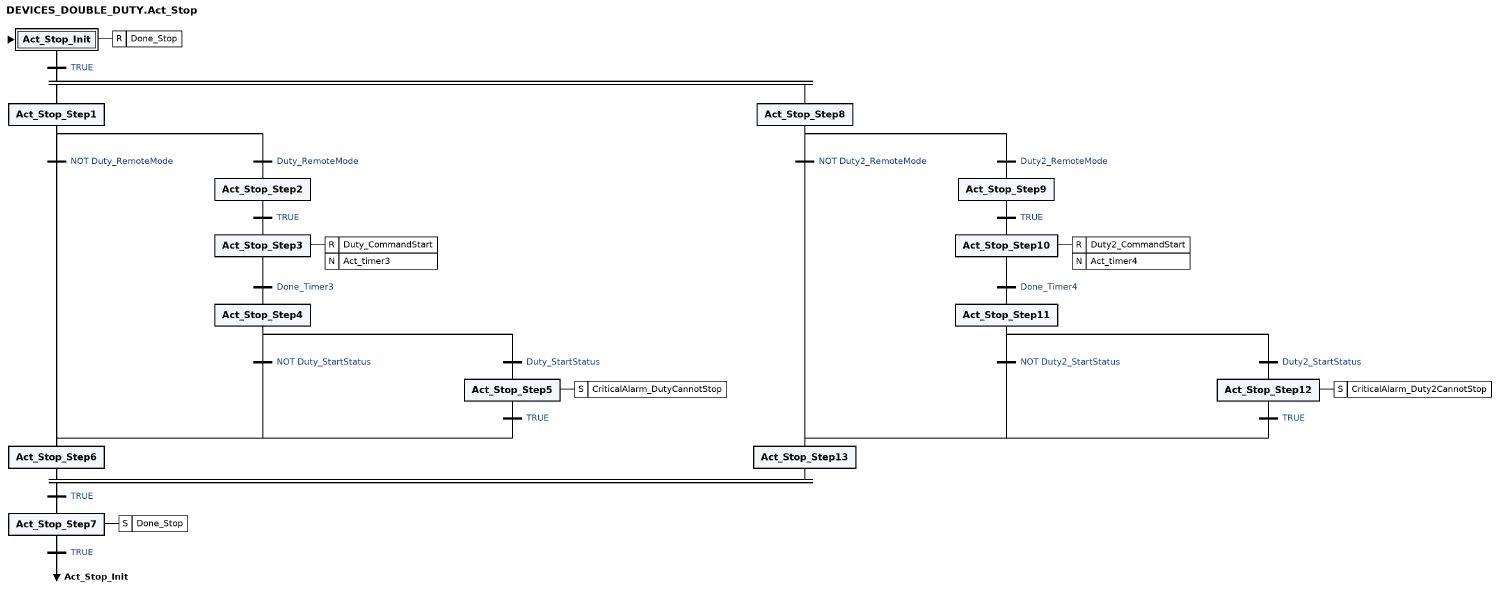
INITIAL_STEP Act_Stop_Init:
	Done_Stop(R);
END_STEP
TRANSITION FROM Act_Stop_Init TO (Act_Stop_Step1, Act_Stop_Step8) := TRUE;
END_TRANSITION
STEP Act_Stop_Step1:
END_STEP
TRANSITION FROM Act_Stop_Step1 TO Act_Stop_Step6 := NOT Duty_RemoteMode;
END_TRANSITION
TRANSITION FROM Act_Stop_Step1 TO Act_Stop_Step2 := Duty_RemoteMode;
END_TRANSITION
STEP Act_Stop_Step2:
END_STEP
TRANSITION FROM Act_Stop_Step2 TO Act_Stop_Step3 := TRUE;
END_TRANSITION
STEP Act_Stop_Step3:
	Duty_CommandStart(R);
	Act_timer3(N);
END_STEP
TRANSITION FROM Act_Stop_Step3 TO Act_Stop_Step4 := Done_Timer3;
END_TRANSITION
STEP Act_Stop_Step4:
END_STEP
TRANSITION FROM Act_Stop_Step4 TO Act_Stop_Step6 := NOT Duty_StartStatus;
END_TRANSITION
TRANSITION FROM Act_Stop_Step4 TO Act_Stop_Step5 := Duty_StartStatus;
END_TRANSITION
STEP Act_Stop_Step5:
	CriticalAlarm_DutyCannotStop(S);
END_STEP
TRANSITION FROM Act_Stop_Step5 TO Act_Stop_Step6 := TRUE;
END_TRANSITION
STEP Act_Stop_Step6:
END_STEP
STEP Act_Stop_Step8:
END_STEP
TRANSITION FROM Act_Stop_Step8 TO Act_Stop_Step13 := NOT Duty2_RemoteMode;
END_TRANSITION
TRANSITION FROM Act_Stop_Step8 TO Act_Stop_Step9 := Duty2_RemoteMode;
END_TRANSITION
STEP Act_Stop_Step9:
END_STEP
TRANSITION FROM Act_Stop_Step9 TO Act_Stop_Step10 := TRUE;
END_TRANSITION
STEP Act_Stop_Step10:
	Duty2_CommandStart(R);
	Act_timer4(N);
END_STEP
TRANSITION FROM Act_Stop_Step10 TO Act_Stop_Step11 := Done_Timer4;
END_TRANSITION
STEP Act_Stop_Step11:
END_STEP
TRANSITION FROM Act_Stop_Step11 TO Act_Stop_Step13 := NOT Duty2_StartStatus;
END_TRANSITION
TRANSITION FROM Act_Stop_Step11 TO Act_Stop_Step12 := Duty2_StartStatus;
END_TRANSITION
STEP Act_Stop_Step12:
	CriticalAlarm_Duty2CannotStop(S);
END_STEP
TRANSITION FROM Act_Stop_Step12 TO Act_Stop_Step13 := TRUE;
END_TRANSITION
STEP Act_Stop_Step13:
END_STEP
TRANSITION FROM (Act_Stop_Step6, Act_Stop_Step13) TO Act_Stop_Step7 := TRUE;
END_TRANSITION
STEP Act_Stop_Step7:
	Done_Stop(S);
END_STEP
TRANSITION FROM Act_Stop_Step7 TO Act_Stop_Init := TRUE;
END_TRANSITION
END_ACTION
ACTION Act_Timer:
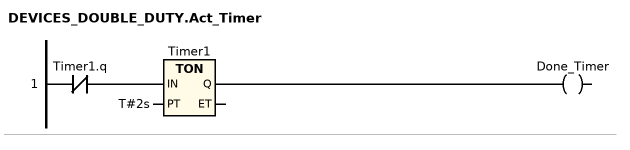
_LD_ (* Ladder Diagram *)
NETWORK 1
	[/Timer1.q] - Timer1:TON(IN: *, PT: T#2s) --- (Done_Timer)
_END_LD_
(* the same logic as Structured Text *)
(* Network 1 *)
Timer1(IN := NOT Timer1.q, PT := T#2s);
Done_Timer := Timer1.Q;
END_ACTION
ACTION Act_Timer2:
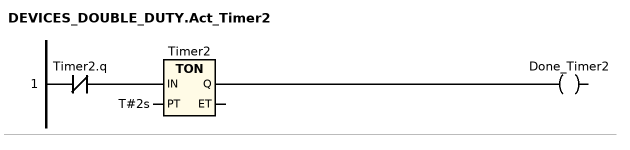
_LD_ (* Ladder Diagram *)
NETWORK 1
	[/Timer2.q] - Timer2:TON(IN: *, PT: T#2s) --- (Done_Timer2)
_END_LD_
(* the same logic as Structured Text *)
(* Network 1 *)
Timer2(IN := NOT Timer2.q, PT := T#2s);
Done_Timer2 := Timer2.Q;
END_ACTION
ACTION Act_Timer3:
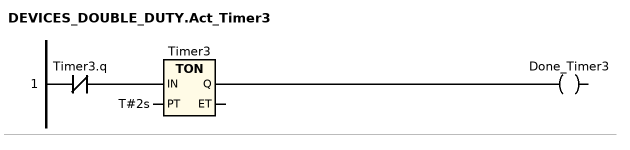
_LD_ (* Ladder Diagram *)
NETWORK 1
	[/Timer3.q] - Timer3:TON(IN: *, PT: T#2s) --- (Done_Timer3)
_END_LD_
(* the same logic as Structured Text *)
(* Network 1 *)
Timer3(IN := NOT Timer3.q, PT := T#2s);
Done_Timer3 := Timer3.Q;
END_ACTION
ACTION Act_Timer4:
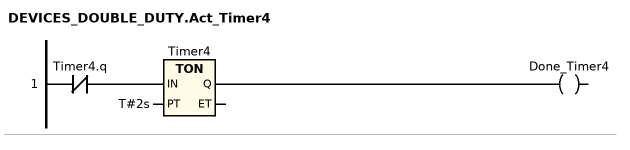
_LD_ (* Ladder Diagram *)
NETWORK 1
	[/Timer4.q] - Timer4:TON(IN: *, PT: T#2s) --- (Done_Timer4)
_END_LD_
(* the same logic as Structured Text *)
(* Network 1 *)
Timer4(IN := NOT Timer4.q, PT := T#2s);
Done_Timer4 := Timer4.Q;
END_ACTION

(* POU test, ST *)
FUNCTION_BLOCK test
VAR_INPUT
END_VAR
VAR_OUTPUT
END_VAR
VAR
	test : ARRAY [0..99] OF INT;
	x: INT;
END_VAR
(*
FOR x:= 0 TO 99 DO
test[x] := 99;
END_FOR
*);
END_FUNCTION_BLOCK

(* POU REUSE_WATER_SYS, SFC *)
FUNCTION_BLOCK REUSE_WATER_SYS
VAR_INPUT
END_VAR
VAR_OUTPUT
END_VAR
VAR
	VacumPump_AB : DEVICES_DUTY_STANDBY;
	LeadPump_AB : DEVICES_DOUBLE_DUTY;
	LeadPump_CD: DEVICES_DOUBLE_DUTY;
	JockeyPump_AB : DEVICES_DUTY_STANDBY;
	LSL308A AT%I*: BOOL;
	LSH308B AT%I*: BOOL;
	LSL308B AT%I*: BOOL;
	LSH308A AT%I*: BOOL;
	Done_Active: BOOL;
	XV101 AT%Q* : BOOL;
	XV102 AT%Q*: BOOL;
	Done_Vacum_Priming: BOOL;
	Done_On_Pump_Seq: BOOL;
	LSH406 AT%I*: BOOL;
	FSL101 AT%I*: BOOL;
	LSH405 AT%I*: BOOL;
	WaterPressureSensor: LREAL;
	Timer1: TON;
	done_TimerWaterPressure: BOOL;
	Reset_TimerWaterPressure: BOOL;
	WarningAlarm_HighPressure : BOOL;
	Done_stop: BOOL;
	RESET: BOOL;
END_VAR
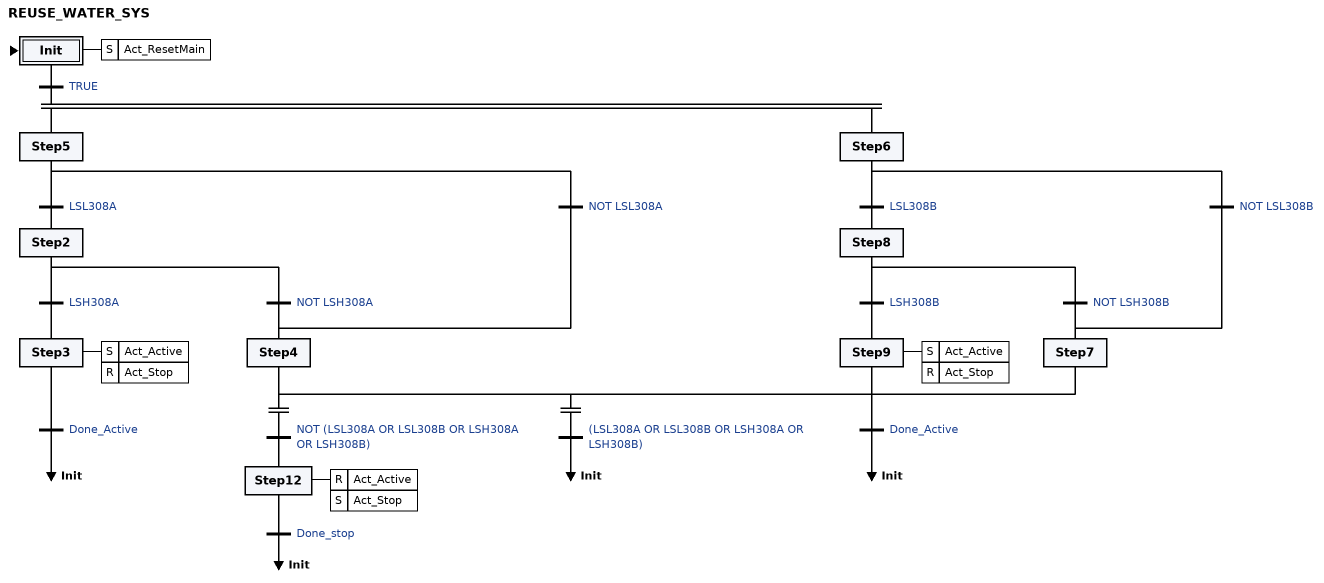
INITIAL_STEP Init:
	Act_ResetMain(S);
END_STEP
TRANSITION FROM Init TO (Step5, Step6) := TRUE;
END_TRANSITION
STEP Step5:
END_STEP
TRANSITION FROM Step5 TO Step2 := LSL308A;
END_TRANSITION
TRANSITION FROM Step5 TO Step4 := NOT LSL308A;
END_TRANSITION
STEP Step2:
END_STEP
TRANSITION FROM Step2 TO Step3 := LSH308A;
END_TRANSITION
TRANSITION FROM Step2 TO Step4 := NOT LSH308A;
END_TRANSITION
STEP Step3:
	Act_Active(S);
	Act_Stop(R);
END_STEP
TRANSITION FROM Step3 TO Init := Done_Active;
END_TRANSITION
STEP Step4:
END_STEP
STEP Step6:
END_STEP
TRANSITION FROM Step6 TO Step8 := LSL308B;
END_TRANSITION
TRANSITION FROM Step6 TO Step7 := NOT LSL308B;
END_TRANSITION
STEP Step8:
END_STEP
TRANSITION FROM Step8 TO Step9 := LSH308B;
END_TRANSITION
TRANSITION FROM Step8 TO Step7 := NOT LSH308B;
END_TRANSITION
STEP Step9:
	Act_Active(S);
	Act_Stop(R);
END_STEP
TRANSITION FROM Step9 TO Init := Done_Active;
END_TRANSITION
STEP Step7:
END_STEP
TRANSITION FROM (Step4, Step7) TO Step12 := NOT (LSL308A OR LSL308B OR LSH308A OR LSH308B);
END_TRANSITION
TRANSITION FROM (Step4, Step7) TO Init := (LSL308A OR LSL308B OR LSH308A OR LSH308B);
END_TRANSITION
STEP Step12:
	Act_Active(R);
	Act_Stop(S);
END_STEP
TRANSITION FROM Step12 TO Init := Done_stop;
END_TRANSITION
END_FUNCTION_BLOCK
ACTION Act_Active:
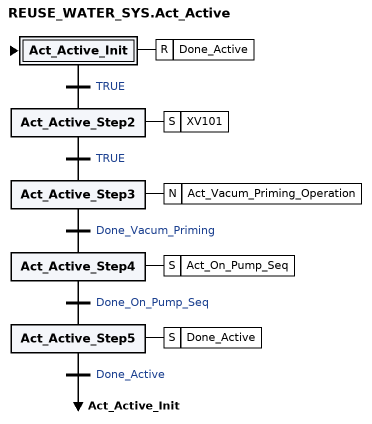
INITIAL_STEP Act_Active_Init:
	Done_Active(R);
END_STEP
TRANSITION FROM Act_Active_Init TO Act_Active_Step2 := TRUE;
END_TRANSITION
STEP Act_Active_Step2:
	XV101(S);
END_STEP
TRANSITION FROM Act_Active_Step2 TO Act_Active_Step3 := TRUE;
END_TRANSITION
STEP Act_Active_Step3:
	Act_Vacum_Priming_Operation(N);
END_STEP
TRANSITION FROM Act_Active_Step3 TO Act_Active_Step4 := Done_Vacum_Priming;
END_TRANSITION
STEP Act_Active_Step4:
	Act_On_Pump_Seq(S);
END_STEP
TRANSITION FROM Act_Active_Step4 TO Act_Active_Step5 := Done_On_Pump_Seq;
END_TRANSITION
STEP Act_Active_Step5:
	Done_Active(S);
END_STEP
TRANSITION FROM Act_Active_Step5 TO Act_Active_Init := Done_Active;
END_TRANSITION
END_ACTION
ACTION Act_JockeyPump_AB_Reset:
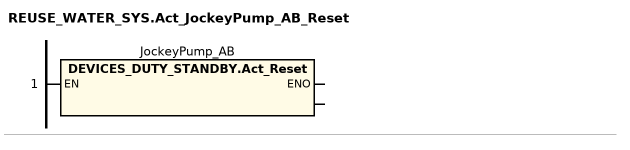
_LD_ (* Ladder Diagram *)
NETWORK 1
	*
		EN --- JockeyPump_AB:DEVICES_DUTY_STANDBY.Act_Reset()
_END_LD_
(* the same logic as Structured Text *)
(* Network 1 *)
JockeyPump_AB();
END_ACTION
ACTION Act_JockeyPump_AB_Start:
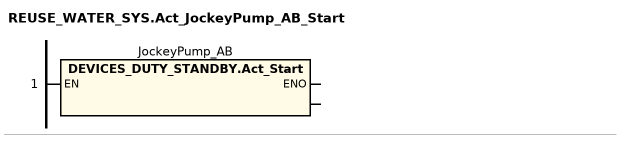
_LD_ (* Ladder Diagram *)
NETWORK 1
	*
		EN --- JockeyPump_AB:DEVICES_DUTY_STANDBY.Act_Start()
_END_LD_
(* the same logic as Structured Text *)
(* Network 1 *)
JockeyPump_AB();
END_ACTION
ACTION Act_JockeyPump_AB_Stop:
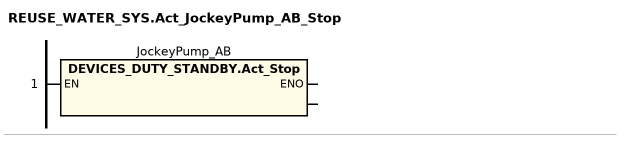
_LD_ (* Ladder Diagram *)
NETWORK 1
	*
		EN --- JockeyPump_AB:DEVICES_DUTY_STANDBY.Act_Stop()
_END_LD_
(* the same logic as Structured Text *)
(* Network 1 *)
JockeyPump_AB();
END_ACTION
ACTION Act_LeadPump_AB_Reset:
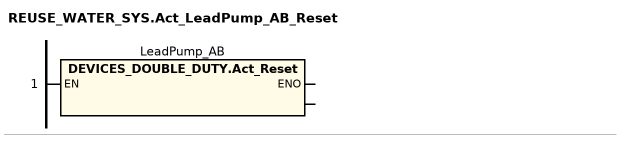
_LD_ (* Ladder Diagram *)
NETWORK 1
	*
		EN --- LeadPump_AB:DEVICES_DOUBLE_DUTY.Act_Reset()
_END_LD_
(* the same logic as Structured Text *)
(* Network 1 *)
LeadPump_AB();
END_ACTION
ACTION Act_LeadPump_AB_Start:
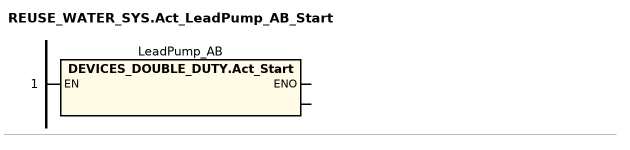
_LD_ (* Ladder Diagram *)
NETWORK 1
	*
		EN --- LeadPump_AB:DEVICES_DOUBLE_DUTY.Act_Start()
_END_LD_
(* the same logic as Structured Text *)
(* Network 1 *)
LeadPump_AB();
END_ACTION
ACTION Act_LeadPump_AB_Stop:
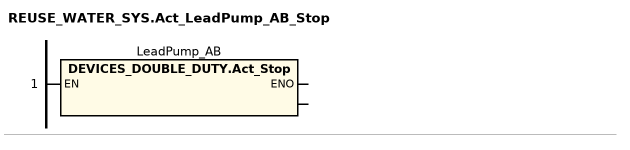
_LD_ (* Ladder Diagram *)
NETWORK 1
	*
		EN --- LeadPump_AB:DEVICES_DOUBLE_DUTY.Act_Stop()
_END_LD_
(* the same logic as Structured Text *)
(* Network 1 *)
LeadPump_AB();
END_ACTION
ACTION Act_LeadPump_CD_Reset:
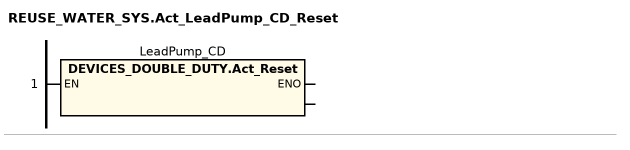
_LD_ (* Ladder Diagram *)
NETWORK 1
	*
		EN --- LeadPump_CD:DEVICES_DOUBLE_DUTY.Act_Reset()
_END_LD_
(* the same logic as Structured Text *)
(* Network 1 *)
LeadPump_CD();
END_ACTION
ACTION Act_LeadPump_CD_Start:
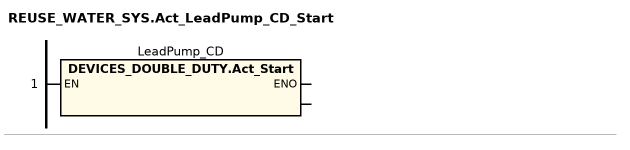
_LD_ (* Ladder Diagram *)
NETWORK 1
	*
		EN --- LeadPump_CD:DEVICES_DOUBLE_DUTY.Act_Start()
_END_LD_
(* the same logic as Structured Text *)
(* Network 1 *)
LeadPump_CD();
END_ACTION
ACTION Act_LeadPump_CD_Stop:
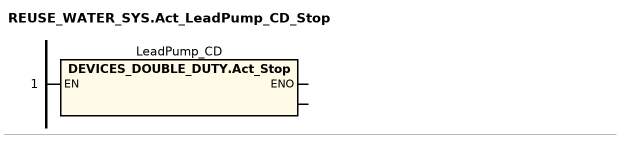
_LD_ (* Ladder Diagram *)
NETWORK 1
	*
		EN --- LeadPump_CD:DEVICES_DOUBLE_DUTY.Act_Stop()
_END_LD_
(* the same logic as Structured Text *)
(* Network 1 *)
LeadPump_CD();
END_ACTION
ACTION Act_On_Pump_Seq:
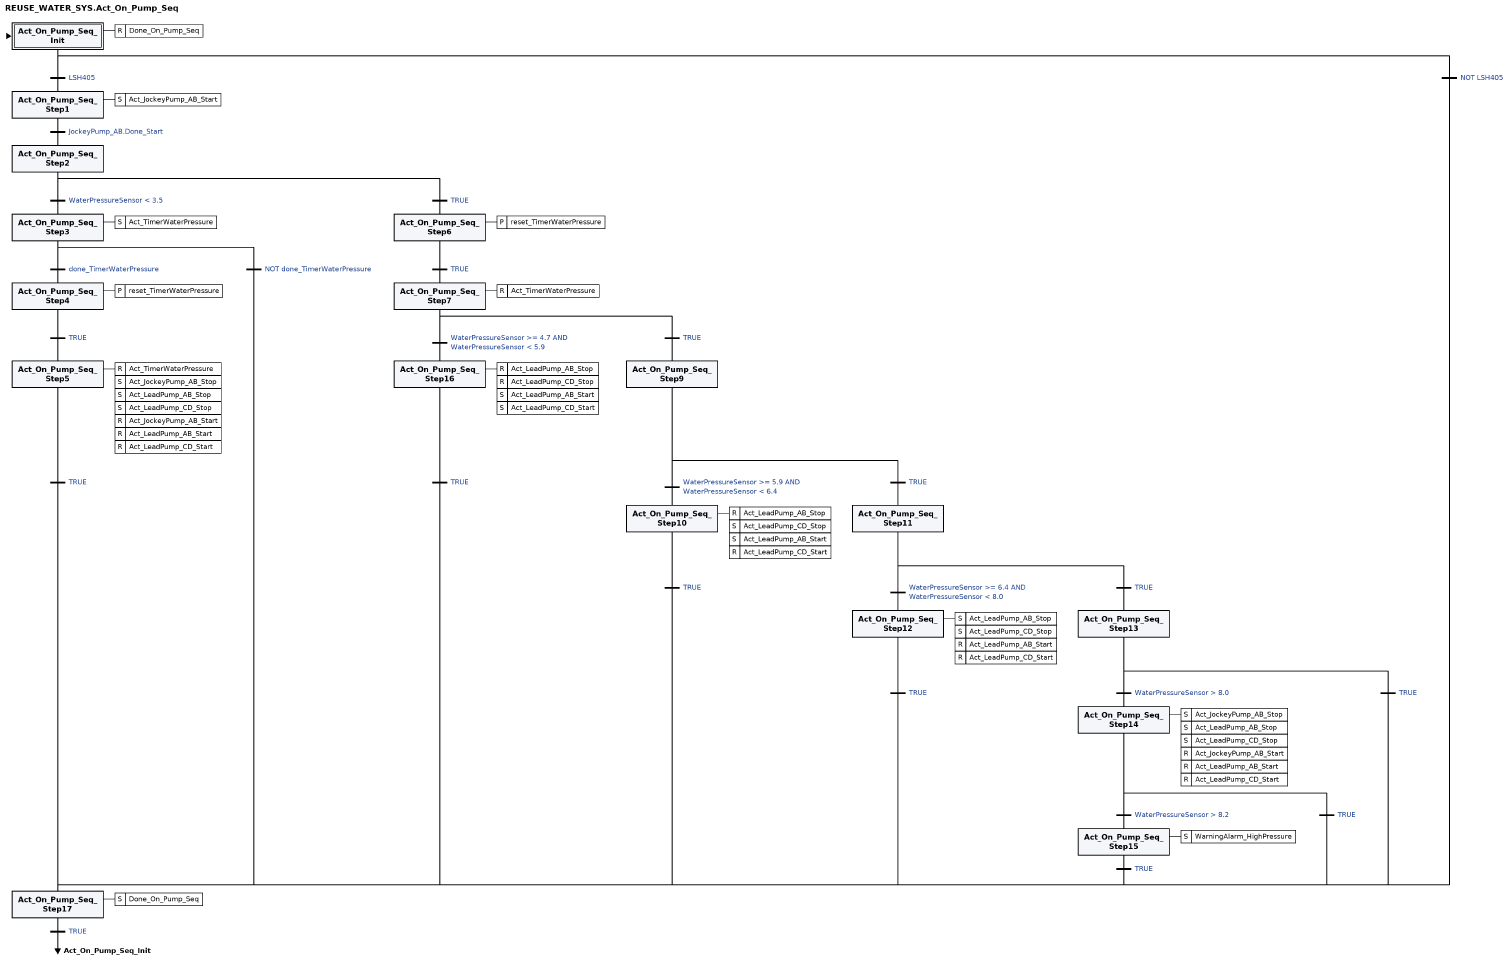
INITIAL_STEP Act_On_Pump_Seq_Init:
	Done_On_Pump_Seq(R);
END_STEP
TRANSITION FROM Act_On_Pump_Seq_Init TO Act_On_Pump_Seq_Step1 := LSH405;
END_TRANSITION
TRANSITION FROM Act_On_Pump_Seq_Init TO Act_On_Pump_Seq_Step17 := NOT LSH405;
END_TRANSITION
STEP Act_On_Pump_Seq_Step1:
	Act_JockeyPump_AB_Start(S);
END_STEP
TRANSITION FROM Act_On_Pump_Seq_Step1 TO Act_On_Pump_Seq_Step2 := JockeyPump_AB.Done_Start;
END_TRANSITION
STEP Act_On_Pump_Seq_Step2:
END_STEP
TRANSITION FROM Act_On_Pump_Seq_Step2 TO Act_On_Pump_Seq_Step3 := WaterPressureSensor < 3.5;
END_TRANSITION
TRANSITION FROM Act_On_Pump_Seq_Step2 TO Act_On_Pump_Seq_Step6 := TRUE;
END_TRANSITION
STEP Act_On_Pump_Seq_Step3:
	Act_TimerWaterPressure(S);
END_STEP
TRANSITION FROM Act_On_Pump_Seq_Step3 TO Act_On_Pump_Seq_Step4 := done_TimerWaterPressure;
END_TRANSITION
TRANSITION FROM Act_On_Pump_Seq_Step3 TO Act_On_Pump_Seq_Step17 := NOT done_TimerWaterPressure;
END_TRANSITION
STEP Act_On_Pump_Seq_Step4:
	reset_TimerWaterPressure(P);
END_STEP
TRANSITION FROM Act_On_Pump_Seq_Step4 TO Act_On_Pump_Seq_Step5 := TRUE;
END_TRANSITION
STEP Act_On_Pump_Seq_Step5:
	Act_TimerWaterPressure(R);
	Act_JockeyPump_AB_Stop(S);
	Act_LeadPump_AB_Stop(S);
	Act_LeadPump_CD_Stop(S);
	Act_JockeyPump_AB_Start(R);
	Act_LeadPump_AB_Start(R);
	Act_LeadPump_CD_Start(R);
END_STEP
TRANSITION FROM Act_On_Pump_Seq_Step5 TO Act_On_Pump_Seq_Step17 := TRUE;
END_TRANSITION
STEP Act_On_Pump_Seq_Step6:
	reset_TimerWaterPressure(P);
END_STEP
TRANSITION FROM Act_On_Pump_Seq_Step6 TO Act_On_Pump_Seq_Step7 := TRUE;
END_TRANSITION
STEP Act_On_Pump_Seq_Step7:
	Act_TimerWaterPressure(R);
END_STEP
TRANSITION FROM Act_On_Pump_Seq_Step7 TO Act_On_Pump_Seq_Step16 := WaterPressureSensor >= 4.7 AND WaterPressureSensor < 5.9;
END_TRANSITION
TRANSITION FROM Act_On_Pump_Seq_Step7 TO Act_On_Pump_Seq_Step9 := TRUE;
END_TRANSITION
STEP Act_On_Pump_Seq_Step16:
	Act_LeadPump_AB_Stop(R);
	Act_LeadPump_CD_Stop(R);
	Act_LeadPump_AB_Start(S);
	Act_LeadPump_CD_Start(S);
END_STEP
TRANSITION FROM Act_On_Pump_Seq_Step16 TO Act_On_Pump_Seq_Step17 := TRUE;
END_TRANSITION
STEP Act_On_Pump_Seq_Step9:
END_STEP
TRANSITION FROM Act_On_Pump_Seq_Step9 TO Act_On_Pump_Seq_Step10 := WaterPressureSensor >= 5.9 AND WaterPressureSensor < 6.4;
END_TRANSITION
TRANSITION FROM Act_On_Pump_Seq_Step9 TO Act_On_Pump_Seq_Step11 := TRUE;
END_TRANSITION
STEP Act_On_Pump_Seq_Step10:
	Act_LeadPump_AB_Stop(R);
	Act_LeadPump_CD_Stop(S);
	Act_LeadPump_AB_Start(S);
	Act_LeadPump_CD_Start(R);
END_STEP
TRANSITION FROM Act_On_Pump_Seq_Step10 TO Act_On_Pump_Seq_Step17 := TRUE;
END_TRANSITION
STEP Act_On_Pump_Seq_Step11:
END_STEP
TRANSITION FROM Act_On_Pump_Seq_Step11 TO Act_On_Pump_Seq_Step12 := WaterPressureSensor >= 6.4 AND WaterPressureSensor < 8.0;
END_TRANSITION
TRANSITION FROM Act_On_Pump_Seq_Step11 TO Act_On_Pump_Seq_Step13 := TRUE;
END_TRANSITION
STEP Act_On_Pump_Seq_Step12:
	Act_LeadPump_AB_Stop(S);
	Act_LeadPump_CD_Stop(S);
	Act_LeadPump_AB_Start(R);
	Act_LeadPump_CD_Start(R);
END_STEP
TRANSITION FROM Act_On_Pump_Seq_Step12 TO Act_On_Pump_Seq_Step17 := TRUE;
END_TRANSITION
STEP Act_On_Pump_Seq_Step13:
END_STEP
TRANSITION FROM Act_On_Pump_Seq_Step13 TO Act_On_Pump_Seq_Step14 := WaterPressureSensor > 8.0;
END_TRANSITION
TRANSITION FROM Act_On_Pump_Seq_Step13 TO Act_On_Pump_Seq_Step17 := TRUE;
END_TRANSITION
STEP Act_On_Pump_Seq_Step14:
	Act_JockeyPump_AB_Stop(S);
	Act_LeadPump_AB_Stop(S);
	Act_LeadPump_CD_Stop(S);
	Act_JockeyPump_AB_Start(R);
	Act_LeadPump_AB_Start(R);
	Act_LeadPump_CD_Start(R);
END_STEP
TRANSITION FROM Act_On_Pump_Seq_Step14 TO Act_On_Pump_Seq_Step15 := WaterPressureSensor > 8.2;
END_TRANSITION
TRANSITION FROM Act_On_Pump_Seq_Step14 TO Act_On_Pump_Seq_Step17 := TRUE;
END_TRANSITION
STEP Act_On_Pump_Seq_Step15:
	WarningAlarm_HighPressure(S);
END_STEP
TRANSITION FROM Act_On_Pump_Seq_Step15 TO Act_On_Pump_Seq_Step17 := TRUE;
END_TRANSITION
STEP Act_On_Pump_Seq_Step17:
	Done_On_Pump_Seq(S);
END_STEP
TRANSITION FROM Act_On_Pump_Seq_Step17 TO Act_On_Pump_Seq_Init := TRUE;
END_TRANSITION
END_ACTION
ACTION Act_ResetMain:
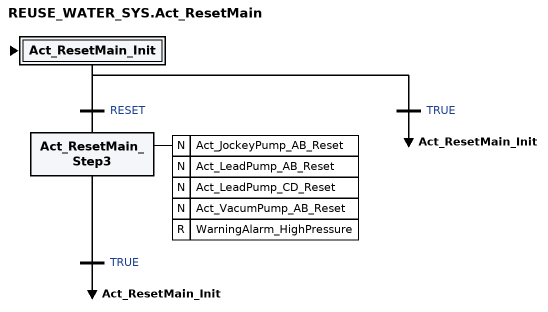
INITIAL_STEP Act_ResetMain_Init:
END_STEP
TRANSITION FROM Act_ResetMain_Init TO Act_ResetMain_Step3 := RESET;
END_TRANSITION
TRANSITION FROM Act_ResetMain_Init TO Act_ResetMain_Init := TRUE;
END_TRANSITION
STEP Act_ResetMain_Step3:
	Act_JockeyPump_AB_Reset(N);
	Act_LeadPump_AB_Reset(N);
	Act_LeadPump_CD_Reset(N);
	Act_VacumPump_AB_Reset(N);
	WarningAlarm_HighPressure(R);
END_STEP
TRANSITION FROM Act_ResetMain_Step3 TO Act_ResetMain_Init := TRUE;
END_TRANSITION
END_ACTION
ACTION Act_Stop:
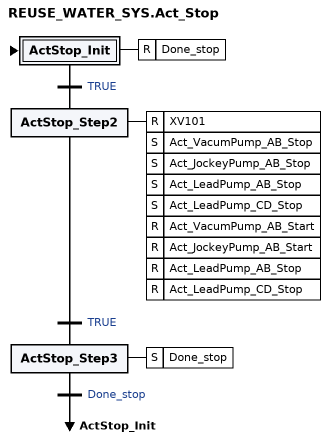
INITIAL_STEP ActStop_Init:
	Done_stop(R);
END_STEP
TRANSITION FROM ActStop_Init TO ActStop_Step2 := TRUE;
END_TRANSITION
STEP ActStop_Step2:
	XV101(R);
	Act_VacumPump_AB_Stop(S);
	Act_JockeyPump_AB_Stop(S);
	Act_LeadPump_AB_Stop(S);
	Act_LeadPump_CD_Stop(S);
	Act_VacumPump_AB_Start(R);
	Act_JockeyPump_AB_Start(R);
	Act_LeadPump_AB_Stop(R);
	Act_LeadPump_CD_Stop(R);
END_STEP
TRANSITION FROM ActStop_Step2 TO ActStop_Step3 := TRUE;
END_TRANSITION
STEP ActStop_Step3:
	Done_stop(S);
END_STEP
TRANSITION FROM ActStop_Step3 TO ActStop_Init := Done_stop;
END_TRANSITION
END_ACTION
ACTION Act_TimerWaterPressure:
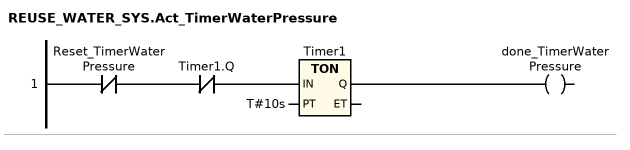
_LD_ (* Ladder Diagram *)
NETWORK 1
	[/Reset_TimerWaterPressure] - [/Timer1.Q] - Timer1:TON(IN: *, PT: T#10s) --- (done_TimerWaterPressure)
_END_LD_
(* the same logic as Structured Text *)
(* Network 1 *)
Timer1(IN := NOT Reset_TimerWaterPressure AND NOT Timer1.Q, PT := T#10s);
done_TimerWaterPressure := Timer1.Q;
END_ACTION
ACTION Act_Vacum_Priming_Operation:
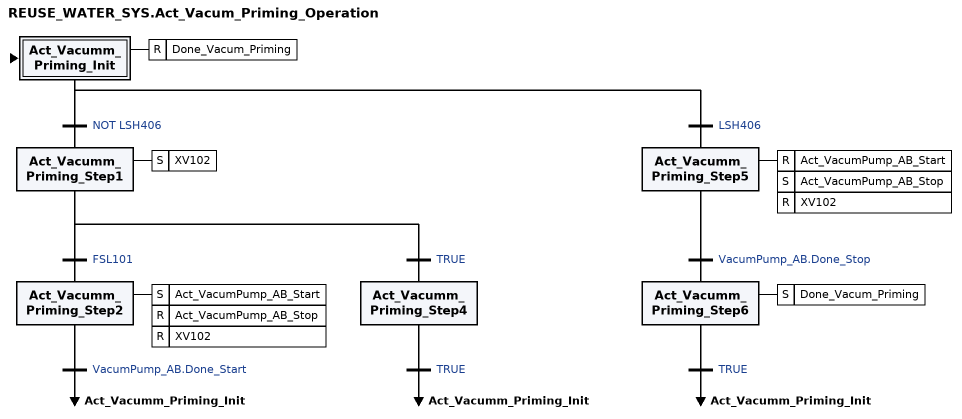
INITIAL_STEP Act_Vacumm_Priming_Init:
	Done_Vacum_Priming(R);
END_STEP
TRANSITION FROM Act_Vacumm_Priming_Init TO Act_Vacumm_Priming_Step1 := NOT LSH406;
END_TRANSITION
TRANSITION FROM Act_Vacumm_Priming_Init TO Act_Vacumm_Priming_Step5 := LSH406;
END_TRANSITION
STEP Act_Vacumm_Priming_Step1:
	XV102(S);
END_STEP
TRANSITION FROM Act_Vacumm_Priming_Step1 TO Act_Vacumm_Priming_Step2 := FSL101;
END_TRANSITION
TRANSITION FROM Act_Vacumm_Priming_Step1 TO Act_Vacumm_Priming_Step4 := TRUE;
END_TRANSITION
STEP Act_Vacumm_Priming_Step2:
	Act_VacumPump_AB_Start(S);
	Act_VacumPump_AB_Stop(R);
	XV102(R);
END_STEP
TRANSITION FROM Act_Vacumm_Priming_Step2 TO Act_Vacumm_Priming_Init := VacumPump_AB.Done_Start;
END_TRANSITION
STEP Act_Vacumm_Priming_Step4:
END_STEP
TRANSITION FROM Act_Vacumm_Priming_Step4 TO Act_Vacumm_Priming_Init := TRUE;
END_TRANSITION
STEP Act_Vacumm_Priming_Step5:
	Act_VacumPump_AB_Start(R);
	Act_VacumPump_AB_Stop(S);
	XV102(R);
END_STEP
TRANSITION FROM Act_Vacumm_Priming_Step5 TO Act_Vacumm_Priming_Step6 := VacumPump_AB.Done_Stop;
END_TRANSITION
STEP Act_Vacumm_Priming_Step6:
	Done_Vacum_Priming(S);
END_STEP
TRANSITION FROM Act_Vacumm_Priming_Step6 TO Act_Vacumm_Priming_Init := TRUE;
END_TRANSITION
END_ACTION
ACTION Act_VacumPump_AB_Reset:
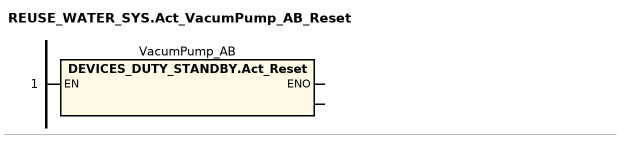
_LD_ (* Ladder Diagram *)
NETWORK 1
	*
		EN --- VacumPump_AB:DEVICES_DUTY_STANDBY.Act_Reset()
_END_LD_
(* the same logic as Structured Text *)
(* Network 1 *)
VacumPump_AB();
END_ACTION
ACTION Act_VacumPump_AB_Start:
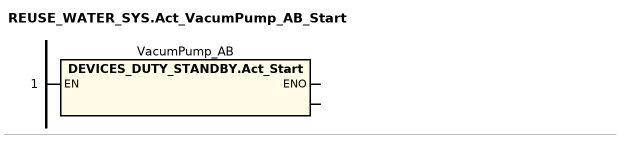
_LD_ (* Ladder Diagram *)
NETWORK 1
	*
		EN --- VacumPump_AB:DEVICES_DUTY_STANDBY.Act_Start()
_END_LD_
(* the same logic as Structured Text *)
(* Network 1 *)
VacumPump_AB();
END_ACTION
ACTION Act_VacumPump_AB_Stop:
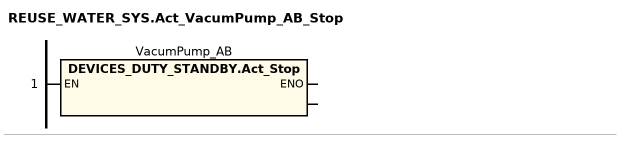
_LD_ (* Ladder Diagram *)
NETWORK 1
	*
		EN --- VacumPump_AB:DEVICES_DUTY_STANDBY.Act_Stop()
_END_LD_
(* the same logic as Structured Text *)
(* Network 1 *)
VacumPump_AB();
END_ACTION

(* POU SCREEN_HOUSE, SFC *)
FUNCTION_BLOCK SCREEN_HOUSE
VAR_INPUT
END_VAR
VAR_OUTPUT
END_VAR
VAR

(*A5*)

	F101x2 AT%I*: BOOL;
	C102x AT %Q*: BOOL;
	C102x_Overload AT%I*: BOOL;
	C102x_Remote AT%I*:  BOOL;
	C102x_StartStatus AT%I*: BOOL;

	ESTOP_ScrewConveyor AT%Q*: BOOL;
	CriticalAlarm_ScrewConveyorCannotStop : BOOL;
	Warning_ScrewCannotStart : BOOL;
	Done_A5_StopScrew: BOOL;
	Done_A5_StartScrewConveyor: BOOL;
(*A6*)
	C101x AT %Q*: BOOL;
	C101x_Remote AT%I*: BOOL;
	C101x_Overload AT%I*: BOOL;
	C101x_StartStatus AT%I*: BOOL;
	XV102x AT%Q*: BOOL;
	Warning_CompactorCannotStart: BOOL;
	Done_A6_StopCompactor: BOOL;
	CriticalAlarm_CompactorCannotStop: BOOL;
	ESTOP_Compactor AT%Q*: BOOL;
	Done_A6_StartCompactor: BOOL;

(*Main*)
	LSH105x AT%I*: BOOL;
	Done_StopF101: BOOL;
	LSHH105x AT%I*: BOOL;
	Done_OpenPS101A1: BOOL;
	Done_A2_StartDuty: BOOL;
	Done_A1_StartDuty: BOOL;
	Done_A1_StartStandby: BOOL;
	done_A2_StartStandby: BOOL;
	Done_A7_On: BOOL;
	Done_A7_Off: BOOL;
	testdone: BOOL;

(*A1*)
	F101x1 AT%I* : BOOL;
	F101x_Remote AT %I*: BOOL;
	F101x1_Overload: BOOL;
	F101x1_StartStatus: BOOL;
	Warning_FineScreenDutyCannotStart: BOOL;
	Done_A4_StartDuty: BOOL;
	Done_A1_StopStandby: BOOL;
	Done_A2_StopStandby: BOOL;
	F101x1_Remote AT %I*: BOOL;
	F101x2_Remote AT %I*: BOOL;
	F101x2_StartStatus: BOOL;
	Done_A4_StartStandby: BOOL;
	Done_A1_StopDuty: BOOL;
	Done_A2_StopDuty: BOOL;
	Warning_FineScreenStandbyCannotStart: BOOL;
END_VAR
